INTERFACE ITF_Base

METHOD GetErrorMessage : String
VAR_INPUT
END_VAR
END_METHOD

METHOD HasError : BOOL
VAR_INPUT
END_VAR
END_METHOD

PROPERTY Name : string
GET
END_GET
END_PROPERTY

END_INTERFACE

(* stored: Version 1.1.0.1, ProductVersion 3.1.4024.12
   Itf ITF_Base: Id {d2e822a2-05f4-4000-9414-c04259fce827}
   Method GetErrorMessage: Id {08153ef1-3ffd-40da-9aec-2cdfc1d0156c}
   Method HasError: Id {e2dbac31-257f-4615-87da-e71e467af487}
   Property Name: Id {01f2294e-8212-4079-a77a-6e90901a0484}
   Get Get: Id {65fdce36-0403-42cf-a9dd-c9d1b6eda0a2} *)
